(* IEC 61131-3 sources: Industry-PLC-LLM/data/PLCBEAD_repo/PLCBEAD_PLCEmbed-main/PLC-BEAD/Source/GEB/TIME_TO_REAL, 1 file *)

(* ---- TIME_TO_REAL.ST ---- *)
FUNCTION TIME_TO_REAL1:REAL

VAR_INPUT
	X :	TIME;
END_VAR

TIME_TO_REAL1 := UDINT_TO_REAL(DINT_TO_UDINT(TIME_TO_DINT(X)));
END_FUNCTION

PROGRAM program0
  VAR
	X :	TIME;
    CEIL5_OUT : REAL;
  END_VAR

  CEIL5_OUT := TIME_TO_REAL1(X);
END_PROGRAM
